{attribute 'GeneratedUsingTerminal: EP2001-1000-0016'}
{attribute addProperty BoxType "EP2001-1000-0016"}
{attribute addProperty Id "WcStateAT %I*BOOL1"}
{attribute addProperty CRC "187373305"}
{attribute addProperty Size "1"}
TYPE WcState_0B2B16F9 :
STRUCT
	{attribute addProperty Name "WcState"}
	WcState AT %I* : BOOL;
END_STRUCT
END_TYPE

(* stored: Version 1.2.0.0, ProductVersion 3.1.4024.9
   DUT WcState_0B2B16F9: Id {131ec781-35d6-40a6-b4bc-c7325d2a9f9e} *)
